FUNCTION_BLOCK AOI_VacuumAdmin
VAR_INPUT
END_VAR
VAR_OUTPUT
END_VAR
VAR_IN_OUT
	admin: UDT_VacuumAdmin;
END_VAR

VAR
	ftVacuum: F_trig;
	tonBlow: TON;
	tonCheck: TON;	
END_VAR

IF admin.i.ActiveIN THEN
	admin.o.ValveIn:=TRUE;
	ELSE 
	admin.o.ValveIn:=FALSE;
END_IF

ftVacuum(CLK:=admin.o.ValveIn , Q=> );
IF ftVacuum.Q THEN
   admin.o.ValveOut:=TRUE;
END_IF
IF tonBlow.Q THEN
   admin.o.ValveOut:=FALSE;
END_IF

tonBlow(IN:=admin.o.ValveOut, PT:=DINT_TO_TIME(admin.i.BlowTime) , Q=> , ET=> );
tonCheck(IN:=admin.o.ValveIn AND NOT admin.i.reset , PT:=DINT_TO_TIME(admin.i.CheckTime)  , Q=> , ET=> );

IF tonCheck.Q AND NOT admin.i.Sensor THEN
	admin.o.Error :=TRUE;
END_IF

IF admin.i.reset THEN
   admin.o.Error :=FALSE;
END_IF

END_FUNCTION_BLOCK

(* stored: Version 1.1.0.1, ProductVersion 3.1.4022.16
   POU AOI_VacuumAdmin: Id {1858a371-e382-42ef-9193-81567ae00b66}, SpecialFunc None *)
